FUNCTION_BLOCK ConvertCommandToString
VAR_INPUT
END_VAR
VAR_OUTPUT
END_VAR
VAR
END_VAR

END_FUNCTION_BLOCK

(* stored: Version 1.1.0.1, ProductVersion 3.1.4022.18
   POU ConvertCommandToString: Id {2416dfc4-341c-4a9a-aa16-3e8ed03ee0bd}, SpecialFunc None *)
